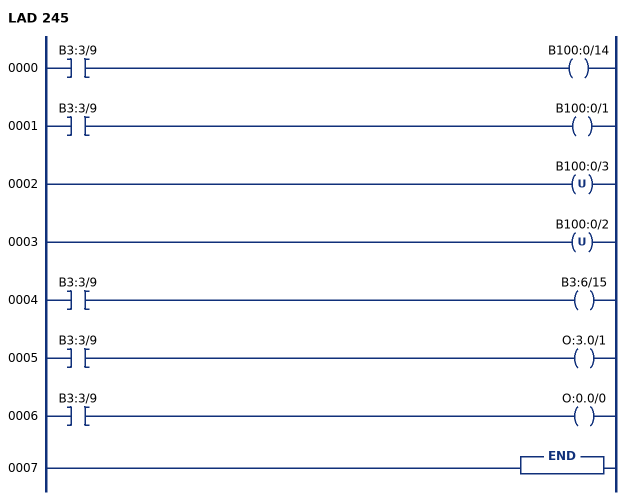
% Rung: 0 %
SOR XIC B3:3/9 OTE B100:0/14 EOR
% Rung: 1 %
SOR XIC B3:3/9 OTE B100:0/1 EOR
% Rung: 2 %
SOR OTU B100:0/3 EOR
% Rung: 3 %
SOR OTU B100:0/2 EOR
% Rung: 4 %
SOR XIC B3:3/9 OTE B3:6/15 EOR
% Rung: 5 %
SOR XIC B3:3/9 OTE O:3.0/1 EOR
% Rung: 6 %
SOR XIC B3:3/9 OTE O:0.0/0 EOR
% Rung: 7 %
SOR END EOR

LADDER 246
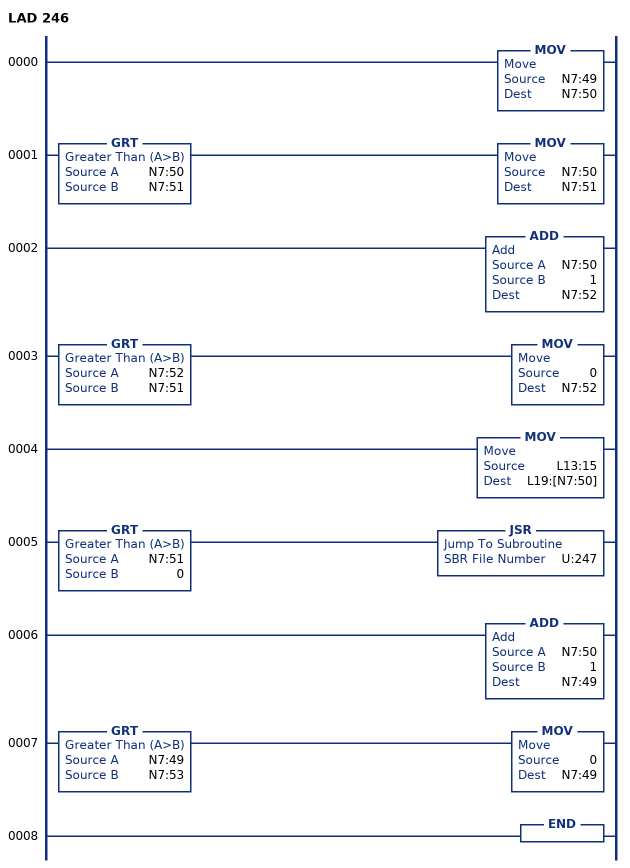
% Rung: 0 %
SOR MOV N7:49 N7:50 EOR
% Rung: 1 %
SOR GRT N7:50 N7:51 MOV N7:50 N7:51 EOR
% Rung: 2 %
SOR ADD N7:50 1 N7:52 EOR
% Rung: 3 %
SOR GRT N7:52 N7:51 MOV 0 N7:52 EOR
% Rung: 4 %
SOR MOV L13:15 L19:[N7:50] EOR
% Rung: 5 %
SOR GRT N7:51 0 JSR U:247 EOR
% Rung: 6 %
SOR ADD N7:50 1 N7:49 EOR
% Rung: 7 %
SOR GRT N7:49 N7:53 MOV 0 N7:49 EOR
% Rung: 8 %
SOR END EOR

LADDER 247
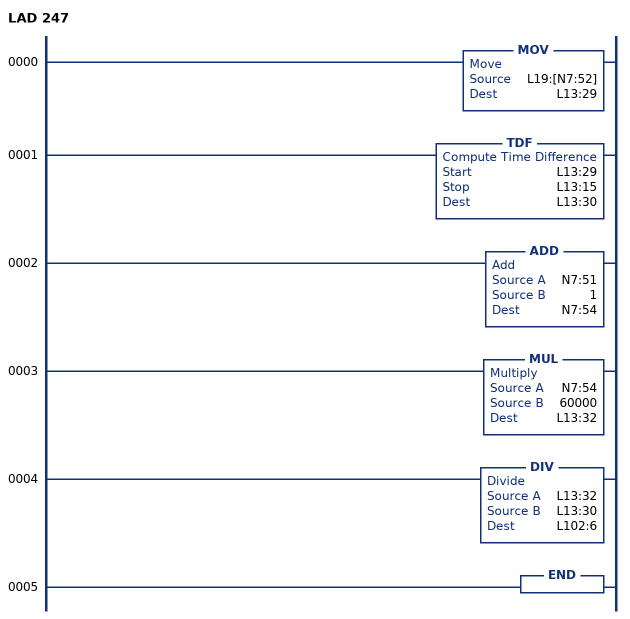
% Rung: 0 %
SOR MOV L19:[N7:52] L13:29 EOR
% Rung: 1 %
SOR TDF L13:29 L13:15 L13:30 EOR
% Rung: 2 %
SOR ADD N7:51 1 N7:54 EOR
% Rung: 3 %
SOR MUL N7:54 60000 L13:32 EOR
% Rung: 4 %
SOR DIV L13:32 L13:30 L102:6 EOR
% Rung: 5 %
SOR END EOR

LADDER 248
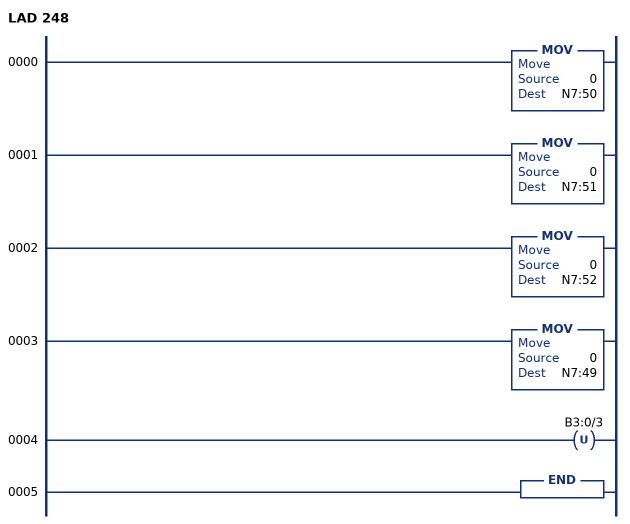
% Rung: 0 %
SOR MOV 0 N7:50 EOR
% Rung: 1 %
SOR MOV 0 N7:51 EOR
% Rung: 2 %
SOR MOV 0 N7:52 EOR
% Rung: 3 %
SOR MOV 0 N7:49 EOR
% Rung: 4 %
SOR OTU B3:0/3 EOR
% Rung: 5 %
SOR END EOR

LADDER 249
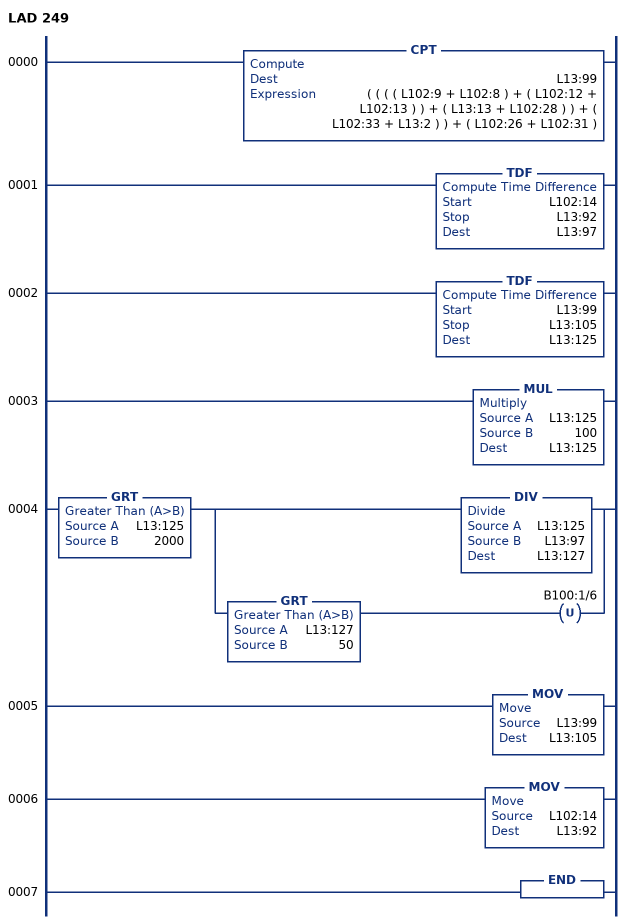
% Rung: 0 %
SOR CPT L13:99 " ( ( ( ( L102:9 + L102:8 ) + ( L102:12 + L102:13 ) ) + ( L13:13 + L102:28 ) ) + ( L102:33 + L13:2 ) ) + ( L102:26 + L102:31 ) " EOR
% Rung: 1 %
SOR TDF L102:14 L13:92 L13:97 EOR
% Rung: 2 %
SOR TDF L13:99 L13:105 L13:125 EOR
% Rung: 3 %
SOR MUL L13:125 100 L13:125 EOR
% Rung: 4 %
SOR GRT L13:125 2000 BST DIV L13:125 L13:97 L13:127 NXB GRT L13:127 50 OTU B100:1/6 BND EOR
% Rung: 5 %
SOR MOV L13:99 L13:105 EOR
% Rung: 6 %
SOR MOV L102:14 L13:92 EOR
% Rung: 7 %
SOR END EOR

LADDER 250
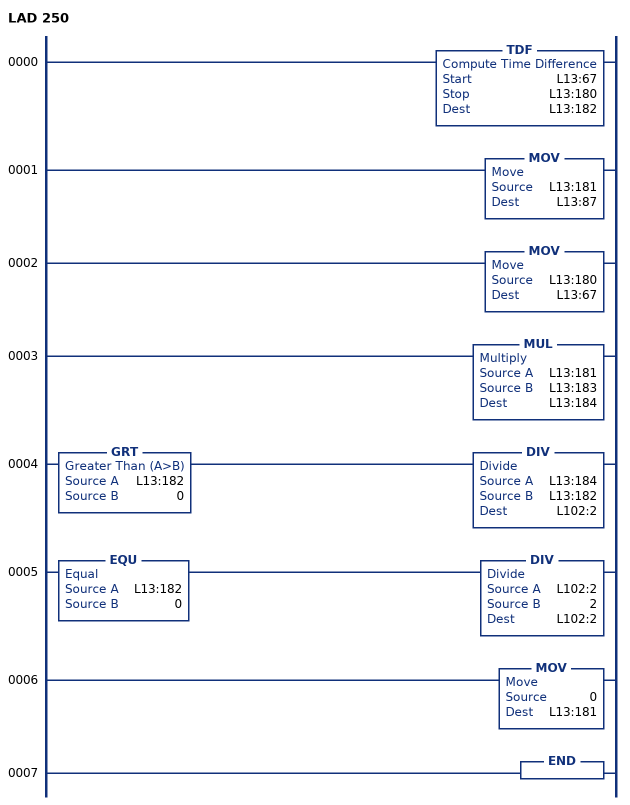
% Rung: 0 %
SOR TDF L13:67 L13:180 L13:182 EOR
% Rung: 1 %
SOR MOV L13:181 L13:87 EOR
% Rung: 2 %
SOR MOV L13:180 L13:67 EOR
% Rung: 3 %
SOR MUL L13:181 L13:183 L13:184 EOR
% Rung: 4 %
SOR GRT L13:182 0 DIV L13:184 L13:182 L102:2 EOR
% Rung: 5 %
SOR EQU L13:182 0 DIV L102:2 2 L102:2 EOR
% Rung: 6 %
SOR MOV 0 L13:181 EOR
% Rung: 7 %
SOR END EOR

LADDER 251
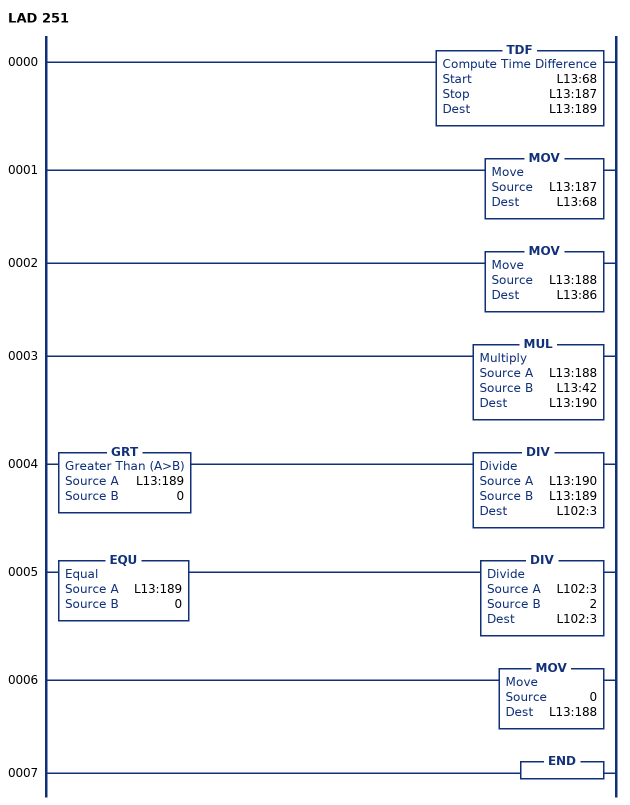
% Rung: 0 %
SOR TDF L13:68 L13:187 L13:189 EOR
% Rung: 1 %
SOR MOV L13:187 L13:68 EOR
% Rung: 2 %
SOR MOV L13:188 L13:86 EOR
% Rung: 3 %
SOR MUL L13:188 L13:42 L13:190 EOR
% Rung: 4 %
SOR GRT L13:189 0 DIV L13:190 L13:189 L102:3 EOR
% Rung: 5 %
SOR EQU L13:189 0 DIV L102:3 2 L102:3 EOR
% Rung: 6 %
SOR MOV 0 L13:188 EOR
% Rung: 7 %
SOR END EOR

LADDER 252
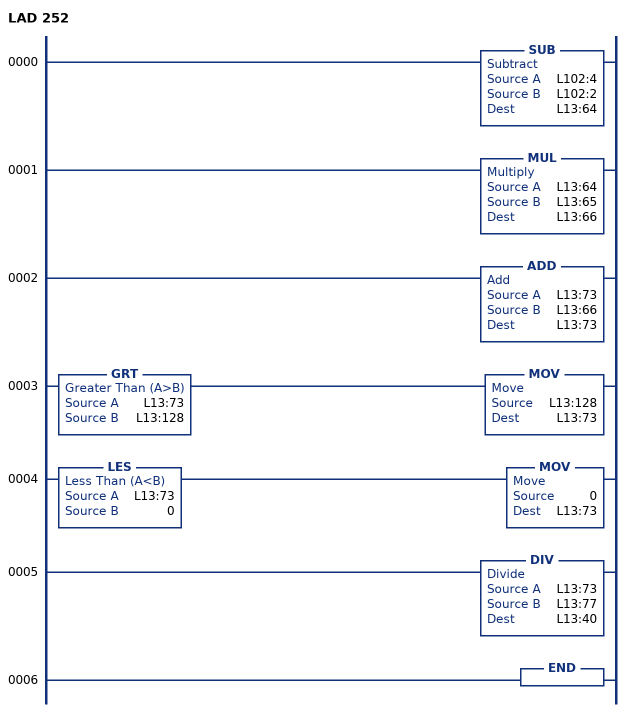
% Rung: 0 %
SOR SUB L102:4 L102:2 L13:64 EOR
% Rung: 1 %
SOR MUL L13:64 L13:65 L13:66 EOR
% Rung: 2 %
SOR ADD L13:73 L13:66 L13:73 EOR
% Rung: 3 %
SOR GRT L13:73 L13:128 MOV L13:128 L13:73 EOR
% Rung: 4 %
SOR LES L13:73 0 MOV 0 L13:73 EOR
% Rung: 5 %
SOR DIV L13:73 L13:77 L13:40 EOR
% Rung: 6 %
SOR END EOR

LADDER 253
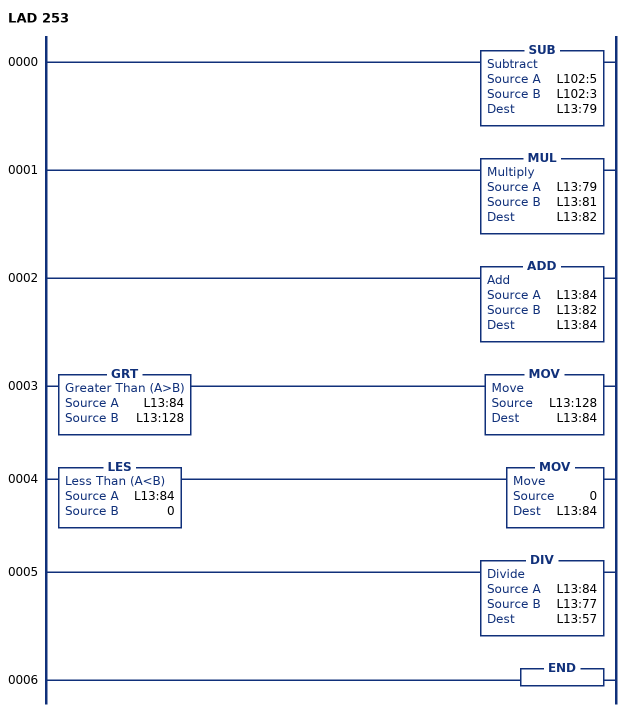
% Rung: 0 %
SOR SUB L102:5 L102:3 L13:79 EOR
% Rung: 1 %
SOR MUL L13:79 L13:81 L13:82 EOR
% Rung: 2 %
SOR ADD L13:84 L13:82 L13:84 EOR
% Rung: 3 %
SOR GRT L13:84 L13:128 MOV L13:128 L13:84 EOR
% Rung: 4 %
SOR LES L13:84 0 MOV 0 L13:84 EOR
% Rung: 5 %
SOR DIV L13:84 L13:77 L13:57 EOR
% Rung: 6 %
SOR END EOR

LADDER 254
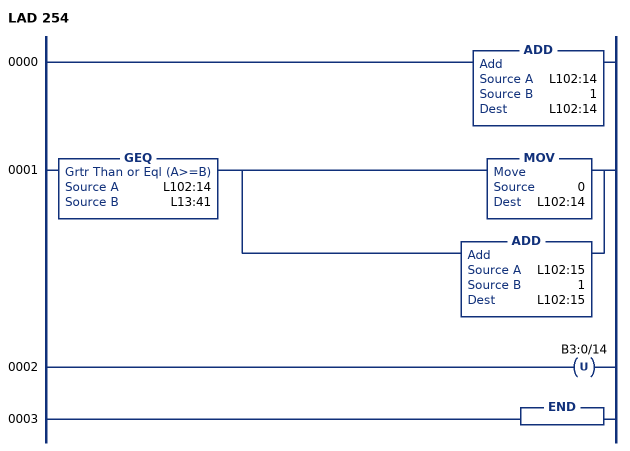
% Rung: 0 %
SOR ADD L102:14 1 L102:14 EOR
% Rung: 1 %
SOR GEQ L102:14 L13:41 BST MOV 0 L102:14 NXB ADD L102:15 1 L102:15 BND EOR
% Rung: 2 %
SOR OTU B3:0/14 EOR
% Rung: 3 %
SOR END EOR

LADDER 255
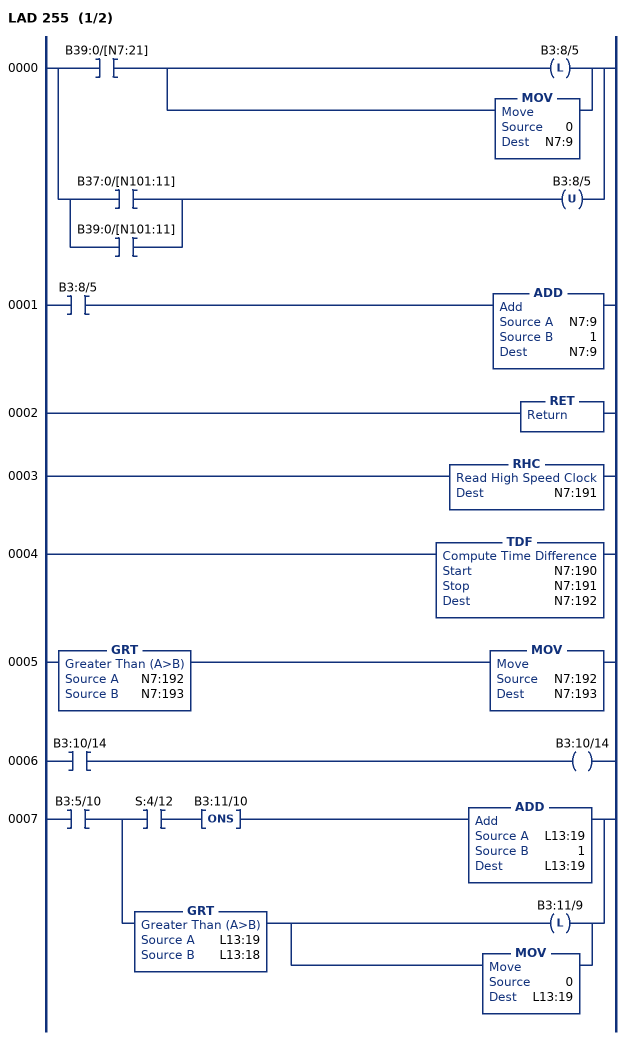
% Rung: 0 %
SOR BST XIC B39:0/[N7:21] BST OTL B3:8/5 NXB MOV 0 N7:9 BND NXB BST XIC B37:0/[N101:11] NXB XIC B39:0/[N101:11] BND OTU B3:8/5 BND EOR
% Rung: 1 %
SOR XIC B3:8/5 ADD N7:9 1 N7:9 EOR
% Rung: 2 %
SOR RET EOR
% Rung: 3 %
SOR RHC N7:191 EOR
% Rung: 4 %
SOR TDF N7:190 N7:191 N7:192 EOR
% Rung: 5 %
SOR GRT N7:192 N7:193 MOV N7:192 N7:193 EOR
% Rung: 6 %
SOR XIC B3:10/14 OTE B3:10/14 EOR
% Rung: 7 %
SOR XIC B3:5/10 BST XIC S:4/12 ONS B3:11/10 ADD L13:19 1 L13:19 NXB GRT L13:19 L13:18 BST OTL B3:11/9 NXB MOV 0 L13:19 BND BND EOR

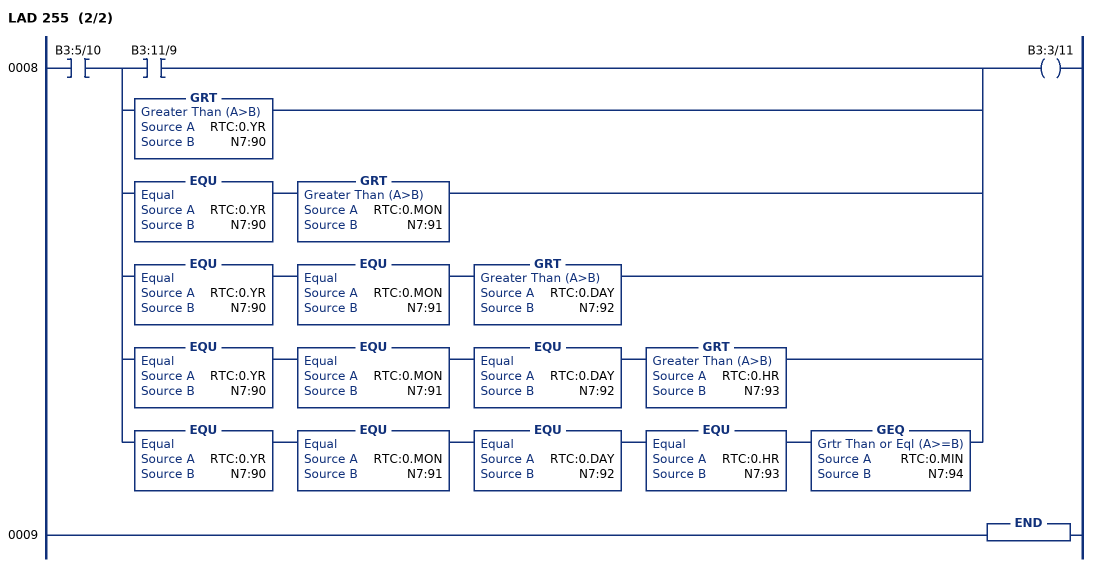
% Rung: 8 %
SOR XIC B3:5/10 BST XIC B3:11/9 NXB GRT RTC:0.YR N7:90 NXB EQU RTC:0.YR N7:90 GRT RTC:0.MON N7:91 NXB EQU RTC:0.YR N7:90 EQU RTC:0.MON N7:91 GRT RTC:0.DAY N7:92 NXB EQU RTC:0.YR N7:90 EQU RTC:0.MON N7:91 EQU RTC:0.DAY N7:92 GRT RTC:0.HR N7:93 NXB EQU RTC:0.YR N7:90 EQU RTC:0.MON N7:91 EQU RTC:0.DAY N7:92 EQU RTC:0.HR N7:93 GEQ RTC:0.MIN N7:94 BND OTE B3:3/11 EOR
% Rung: 9 %
SOR END EOR

DATA TABLE (non-zero values as saved)
DATA B3
% B3:0 % 0XA830 0X0360 0X4001 0X5109 0XCEBB 0X1550 0X0C30 0X0421 0X2F80 0X24B0
% B3:10 % 0X21E4 0X0006 0X2000 0X0000 0X0000 0X0000 0X0000 0X0000 0X0000 0X0000
% B3:50 % 0X0001 0X0000 0X0000 0X0000 0X0000 0X0000 0X0000 0X0000 0X0000 0X0000
DATA T4
% .PRE .ACC %
% T4:0 % 0 2
% T4:1 % 150 0
% T4:2 % 400 0
% T4:3 % 250 87
% T4:4 % 1000 0
% T4:5 % 5 5
% T4:6 % 10 32766
% T4:7 % 1500 0
% T4:8 % 20 11
% T4:9 % 50 21
% T4:10 % 200 200
% T4:11 % 666 419
% T4:12 % 20 20
% T4:13 % 250 0
% T4:14 % 666 0
% T4:15 % 1000 1001
% T4:16 % 400 0
% T4:17 % 100 40
% T4:18 % 5 0
% T4:19 % 300 0
% T4:20 % 200 0
% T4:21 % 200 0
% T4:22 % 200 0
% T4:23 % 250 0
% T4:24 % 666 0
% T4:25 % 666 0
% T4:26 % 666 0
% T4:27 % 250 0
% T4:28 % 250 0
% T4:29 % 5000 0
% T4:30 % 333 0
% T4:31 % 333 17
% T4:32 % 250 112
% T4:33 % 250 80
% T4:34 % 500 0
DATA C5
% .PRE .ACC %
% C5:0 % 32766 0
DATA R6
% .LEN .POS %
% R6:0 % 1250 0
% R6:1 % 1250 0
% R6:2 % 1050 0
% R6:3 % 1050 0
% R6:4 % 1250 0
% R6:5 % 1250 0
% R6:6 % 1713 0
% R6:7 % 1024 0
% R6:8 % 1024 0
% R6:9 % 3 0
% R6:10 % 2048 0
% R6:11 % 2048 0
% R6:12 % 10 0
% R6:13 % 10 0
% R6:14 % 10 0
% R6:15 % 10 0
% R6:16 % 1713 0
% R6:17 % 2048 0
% R6:18 % 2048 0
% R6:19 % 10 0
DATA N7
% N7:0 % 17248 3 1019 137 3 202 0 0 500 0
% N7:10 % 1000 0 0 2 20 20 1000 2000 50 1050
% N7:20 % 0 589 10 4 205 46 0 0 150 250
% N7:30 % 666 1453 150 0 23 1229 77 27 0 27
% N7:40 % 23 15 0 15 125 1223 208 228 501 14
% N7:50 % 13 16 14 16 17 0 0 0 500 0
% N7:60 % 1713 2048 2048 1016 995 985 4999 5 400 400
% N7:70 % 100 200 300 400 90 190 290 390 2832 0
% N7:80 % 1500 0 1249 1258 1261 1271 37 48 0 0
% N7:90 % 2011 4 4 12 1 37 48 222 222 12
% N7:100 % 1003 90 110 100 175 25 0 0 0 0
% N7:190 % 11514 17572 55 88 0 0 0 0 0 0
DATA F8
% F8:0 % 6
DATA L13
% L13:0 % 12177 115617 0 35047 171397
% L13:5 % 5982 75 5982 131379 0
% L13:10 % 0 24586 31497 15 90
% L13:15 % 1271687210 -2147483648 2147483647 2147483647 82058
% L13:20 % 26125172 1947430994 777 38907 100
% L13:25 % 5974 2236 13746 0 1271231348
% L13:30 % 455205 5982 1020000 1265392100 444
% L13:35 % 1 624336 0 0 0
% L13:40 % 14963 1000000000 1000000 1265392072 1270506591
% L13:45 % 1270565467 150 0 28 23904136
% L13:50 % 2987 30027 1261820933 0 0
% L13:55 % 2928 2027255 12170 -1783954998 -1783954972
% L13:60 % 26 104 -1783954986 600 5
% L13:65 % 100 500 209600863 209600861 12
% L13:70 % 1944674498 8 118 1496300 23904136
% L13:75 % 11 60 100 1261820941 2
% L13:80 % 24 74 148 7 1217006
% L13:85 % 396020 178 178 0 2988
% L13:90 % 2929 5 40650 5 1270506619
% L13:95 % 10 714556 0 1270565492 92300
% L13:100 % 300 6 1300 14 503
% L13:105 % 92300 31 25702486 43977 25702480
% L13:110 % 6 100 50 1947010411 1947034989
% L13:115 % 1947034997 8 4 1947034993 26
% L13:120 % 0 3744 50 100 10
% L13:125 % 0 1944674498 2147483647 3276500 420618
% L13:130 % 2 2 0 99 0
% L13:135 % 0 0 396032 5 70
% L13:140 % 0 5 36 50 50
% L13:145 % 30028 5 5 5 11
% L13:150 % 12 20 10840 -10840 24586
% L13:155 % 0 -10 0 0 4589052
% L13:160 % 10 28 25 1220 45
% L13:165 % 1947014454 1947035226 1947014454 1947035226 6706
% L13:170 % 12817 10838 10608 500 300
% L13:175 % 4 4 42 23 38
% L13:180 % 209616706 55 50937 1000000 178000000
% L13:185 % 0 1 209616866 56 50879
% L13:190 % 178000000 0 0 0 0
DATA L19
% L19:0 % 1271235868 1271237376 1271238884 1271240392 1271241901
% L19:5 % 1271243407 1271244912 1271246421 1271247926 1271249435
% L19:10 % 1271260473 1271261980 1271263488 1271264994 1271231348
% L19:15 % 1271232856 1271234362 0 0 0
DATA L20
% L20:0 % 1270131466 1270133482 1270135505 1270137523 1270139540
% L20:5 % 1270141561 1270143575 1270145595 1270147612 1270149631
% L20:10 % 1270151647 1270153666 1270155686 1270157705 1270159721
% L20:15 % 1270161739 1270163756 1270165777 1270167792 1270371104
% L20:20 % 1270384685 1270421471 1270421727 1270422998 1270423254
% L20:25 % 1270424529 1270424784 1270427199 1270427454 1270427709
% L20:30 % 1270427962 1270428216 1270437435 1270448135 1270456656
% L20:35 % 1270465035 1270495753 1270506591 1270107259 1270109275
% L20:40 % 1270111291 1270113305 1270115322 1270117343 1270119362
% L20:45 % 1270121381 1270123395 1270125412 1270127434 1270129451
DATA L21
% L21:0 % 1946882098 1946882810 1946883524 1946884236 1946884947
% L21:5 % 1946885660 1946886371 1946887084 1946887795 1946888507
% L21:10 % 1946889218 1946889931 1946890644 1946891356 1946892067
% L21:15 % 1946892779 1946893491 1946894204 1946894915 1946966646
% L21:20 % 1946971438 1946984417 1946984507 1946984956 1946985046
% L21:25 % 1946985496 1946985586 1946986439 1946986529 1946986619
% L21:30 % 1946986708 1946986798 1946990050 1946993825 1946996833
% L21:35 % 1946999790 1947010630 1947014454 1946873557 1946874268
% L21:40 % 1946874979 1946875690 1946876402 1946877115 1946877827
% L21:45 % 1946878540 1946879251 1946879963 1946880676 1946881387
DATA L22
% L22:0 % 1257481069 1257490512 1257498604 1257509115 1257516794
% L22:5 % 1257567664 1257592269 1257599923 1257608372 1257615862
% L22:10 % 1257623940 1257637265 1257644499 1257651980 1263850422
% L22:15 % 1263850676 1263850931 1263851185 1263851438 1263851693
% L22:20 % 1263851947 1263852201 1263900246 1263911293 1263922536
% L22:25 % 1263934034 1263944967 1263982469 1264000818 1264012035
% L22:30 % 1264029664 1264041339 1264683787 1265398338 1266216256
% L22:35 % 1266227865 1266238397 1266246323 1266255854 1266263826
% L22:40 % 1266271246 1266279054 1266286959 1270517200 1270525795
% L22:45 % 1270534031 1270546070 1270554859 1270565467 1257463793
DATA L23
% L23:0 % 1942933757 1942937564 1942940828 1942945066 1942948162
% L23:5 % 1942968675 1942978596 1942981682 1942985089 1942988109
% L23:10 % 1942991367 1942996739 1942999655 1943002672 1944674498
% L23:15 % 1944674498 1944674498 1944674498 1944674498 1944674498
% L23:20 % 1944674498 1944674498 1944683647 1944687544 1944691511
% L23:25 % 1944695567 1944699425 1944712657 1944719131 1944723087
% L23:30 % 1944729306 1944733424 1944960087 1945212191 1945500760
% L23:35 % 1945504856 1945508572 1945511368 1945514730 1945517543
% L23:40 % 1945520161 1945522916 1945525705 1947018197 1947021229
% L23:45 % 1947024134 1947028382 1947031482 1947035226 1942926789
DATA L30
% L30:0 % 1097513510 1097513738 1097513967 1097514196 1097514426
% L30:5 % 1097514655 1097514883 1097515111 1097515339 1188692931
% L30:10 % 1263848224 1263850325 1263850578 1263851854 1263852108
% L30:15 % 1263883310 1263893977 1263905023 1263916268 1263927766
% L30:20 % 1263938694 1263976204 1263994554 1264005760 1264023393
% L30:25 % 1264035071 1264677516 1265392072 1071309024 1071309250
% L30:30 % 1071309476 1071429569 1071429795 1071431153 1071431379
% L30:35 % 1071431606 1088333039 1088333266 1088334623 1088334848
% L30:40 % 1088335075 1089808842 1089809070 1089810430 1089810657
% L30:45 % 1089810882 1092780028 1092791426 1092806921 1097513283
DATA L31
% L31:0 % 3522828 3522897 3522967 3523035 3523105
% L31:5 % 3523175 3523244 3523313 3523382 20590662
% L31:10 % 23368545 23368545 23368545 23368545 23368545
% L31:15 % 23371832 23375594 23379493 23383460 23387517
% L31:20 % 23391373 23404607 23411081 23415034 23421255
% L31:25 % 23425375 23652030 23904136 2077757 2077757
% L31:30 % 2077757 2077757 2077757 2077757 2077757
% L31:35 % 2077757 2077757 2077757 2077757 2077757
% L31:40 % 2077757 2077757 2077757 2077757 2077757
% L31:45 % 2077757 2091375 2094821 2099507 3522760
DATA L32
% L32:0 % 1257480992 1257490438 1257498530 1257509041 1257516717
% L32:5 % 1257567592 1257592195 1257599851 1257608295 1257615790
% L32:10 % 1257623864 1257637189 1257644427 1257651905 1261820430
% L32:15 % 1261820933 1256830919 1256831425 1256831932 1256832439
% L32:20 % 1256832946 1256840038 1256920077 1256920583 1256921090
% L32:25 % 1256921596 1256922103 1256938651 1256948212 1256956941
% L32:30 % 1256965556 1256986583 1256995787 1257004741 1257012938
% L32:35 % 1257029359 1257047788 1257056336 1257091378 1257111913
% L32:40 % 1257128874 1257152815 1257160372 1257191338 1257205037
% L32:45 % 1257400333 1257427641 1257445460 1257455539 1257463721
DATA L33
% L33:0 % 1942933726 1942937534 1942940798 1942945036 1942948131
% L33:5 % 1942968646 1942978566 1942981653 1942985058 1942988080
% L33:10 % 1942991336 1942996708 1942999626 1943002642 1944674498
% L33:15 % 1944674498 1942682094 1942682278 1942682462 1942682645
% L33:20 % 1942682829 1942685403 1942714449 1942714633 1942714817
% L33:25 % 1942715001 1942715185 1942721190 1942724660 1942727827
% L33:30 % 1942730953 1942738585 1942741925 1942745174 1942748150
% L33:35 % 1942754110 1942759038 1942762486 1942776618 1942784898
% L33:40 % 1942791737 1942801391 1942804438 1942816923 1942822448
% L33:45 % 1942901198 1942912211 1942919397 1942923461 1942926760
DATA B100
% B100:0 % 0X2780 0X00A0 0X0004 0X0000 0X0000 0X0000 0X0000 0X0000 0X0000 0X0000
DATA N101
% N101:0 % 114 0 0 0 1183 100 1015 1200 1220 1238
% N101:10 % 1248 1604 10 16383 1269 17365 3010 250 333 333
% N101:20 % 1000 500 400 0 0 0 250 250 0 0
DATA L102
% L102:0 % 20 10 3507 3503 3500
% L102:5 % 3500 2 11 0 0
% L102:10 % -10840 129 0 0 40650
% L102:15 % 0 30 10 30 10
% L102:20 % 0 5 76747 0 28
% L102:25 % 28 0 3 81649 0
% L102:30 % 8 0 13 10636 3
% L102:35 % 174 302 0 999999 25
% L102:40 % 0 3 0 0 0
